// TIA Portal V19 export
FUNCTION_BLOCK "CpuPreviuosCycleTime"   // FB4, LAD
TITLE = Cpu Previus cycle time / Get CPU Previous Cycle Time
// stored: Access Published, MemoryReserve 100, SetENOAutomatically false
   VAR_OUTPUT
      PrevCycleTime : Int;
   END_VAR
   VAR
      CpuDateTime { ExternalAccessible := 'False'; ExternalVisible := 'False'; ExternalWritable := 'False'} : Date_And_Time;
      PrevCpuDateTime : Date_And_Time;
      LastCpuCycleTime : Time;
   END_VAR
   VAR_TEMP
      Ret : Int;
   END_VAR
BEGIN

REGION Network 1 (SCL): Previus cycle time calculated with cpu time / Main
   #Ret := RD_SYS_T(OUT => #CpuDateTime);

   IF "Sys".FirstPLCCycle THEN
       #PrevCpuDateTime := #CpuDateTime;
   END_IF;

   #LastCpuCycleTime := T_DIFF(IN1 := #CpuDateTime, IN2 := #PrevCpuDateTime);

   IF #LastCpuCycleTime <= T#0MS THEN
       #LastCpuCycleTime := T#1MS;
   END_IF;

   #PrevCpuDateTime := #CpuDateTime;
   #PrevCycleTime := TIME_TO_INT(#LastCpuCycleTime);
END_REGION
END_FUNCTION_BLOCK
